{attribute 'qualified_only'}
{attribute 'strict'}
TYPE E_CircleWriteStep :
(
	Check,
	First_Potision_Move,
	Write_Circle,
	Z_Axix_Up_Potision
);
END_TYPE

(* stored: Version 1.1.0.1, ProductVersion 3.1.4024.12
   DUT E_CircleWriteStep: Id {3606e005-34c4-4043-a04d-866e9517e1a7} *)
